// TIA Portal V18 export
DATA_BLOCK "Alarms_DB"   // DB9
// stored: InstanceOfName Alarms, InstanceOfType FB
"Alarms"
   // VAR
   //    BypassTempAlarm_TON { S7_SetPoint := 'True'} : TON_TIME;
   //    TDPressTxFaul_TON { S7_SetPoint := 'True'} : TON_TIME;
   //    HiTemp_TON { S7_SetPoint := 'True'} : TON_TIME;
   //    NoFlushFlow_TON { S7_SetPoint := 'True'} : TON_TIME;
   //    ChargeFault_TON { S7_SetPoint := 'True'} : TON_TIME;
   //    HiTempRPM_TON { S7_SetPoint := 'True'} : TON_TIME;
   //    HornOn_TP { S7_SetPoint := 'True'} : TP_TIME;
   //    HiTempAlarm_TON { S7_SetPoint := 'True'} : TON_TIME;
   //    FlushFault_TP { S7_SetPoint := 'True'} : TP_TIME;
   //    LubeFlowFault_TON { S7_SetPoint := 'True'} : TON_TIME;
   //    LubeFault_TP { S7_SetPoint := 'True'} : TP_TIME;
   //    Charge2Fault_TON { S7_SetPoint := 'True'} : TON_TIME;
   //    Charge1Fault_TP { S7_SetPoint := 'True'} : TP_TIME;
   //    Charge2Fault_TP { S7_SetPoint := 'True'} : TP_TIME;
   //    FilterFault_TP { S7_SetPoint := 'True'} : TP_TIME;
   //    AuxPumpFault_TP { S7_SetPoint := 'True'} : TP_TIME;
   //    FanFault_TP { S7_SetPoint := 'True'} : TP_TIME;
   //    M1Fault_TP { S7_SetPoint := 'True'} : TP_TIME;
   //    M2Fault_TP { S7_SetPoint := 'True'} : TP_TIME;
   //    HiTempFault_TP { S7_SetPoint := 'True'} : TP_TIME;
   //    TankLevelFault_TP { S7_SetPoint := 'True'} : TP_TIME;
   //    TankTempFault_TP { S7_SetPoint := 'True'} : TP_TIME;
   //    HiTempShtdwn_TP { S7_SetPoint := 'True'} : TP_TIME;
   //    TDPressTXFault_TP { S7_SetPoint := 'True'} : TP_TIME;
   //    EngineFault_TP { S7_SetPoint := 'True'} : TP_TIME;
   //    BypassHiTemp_Tp { S7_SetPoint := 'True'} : TP_TIME;
   //    ComFault_Tp { S7_SetPoint := 'True'} : TP_TIME;
   //    SystemFault_Tp { S7_SetPoint := 'True'} : TP_TIME;
   // END_VAR
BEGIN
END_DATA_BLOCK
